FUNCTION Func_InRange : Bool
VAR_INPUT
	IstPos 	:REAL;
	SollPos	:REAL;
	Fenster	:REAL := 0.5;
END_VAR

 Func_InRange := 	IstPos > SollPos - Fenster
 					AND IstPos < SollPos + Fenster;

END_FUNCTION

(* stored: Version 1.1.0.1
   POU Func_InRange: Id {b8543b1a-e673-418b-9c50-ee94aa129029}, SpecialFunc None *)
